(* PLC project Tc2_Utilities.GUID_TO_REGSTRING Demo, tc3-libraries-kb TwinCAT 3.1 *)
(* stored: creationDateTime 2026-05-12T10:00:00, modificationDateTime 2026-05-12T10:00:00 *)

PROGRAM P_Demo_GUID_TO_REGSTRING
  VAR
    gMachineUniqueId : GUID;  (* 从 BIOS / dongle 读到的机器唯一 ID *)
    sRegistryFormatId : STRING;  (* 写到 Windows 注册表的带花括号 GUID 串 *)
    bFormatRequest : BOOL;  (* 在线置 TRUE 触发一次格式化 *)
  END_VAR

// =============================================================================
// 场景：工业 PC 启动时把 BIOS / dongle 读到的机器唯一 ID 写到 Windows
//       注册表项 HKLM\SOFTWARE\Plant\MachineId，便于其他 Windows 服务
//       （如 OPC UA Server）通过 RegEdit 读到统一标识。
// 价值：注册表 / WMI 习惯用 '{...}' 包裹 GUID；本函数一行得到，免去
//       CONCAT('{', GUID_TO_STRING(g), '}') 三步拼接。
// 验证步骤：
//   1. 登录后 gMachineUniqueId 各字段全 0，sRegistryFormatId = ''。
//   2. 在线设置 gMachineUniqueId.Data1 := 16#12345678; .Data2 := 16#1234;
//      .Data3 := 16#5678; .Data4 := [16#9A,16#BC,16#DE,16#F0,16#12,16#34,16#56,16#78];
//   3. 写 bFormatRequest := TRUE。
//   4. 观察 sRegistryFormatId = '{12345678-1234-5678-9ABC-DEF012345678}'
//      （长度 38，含花括号，hex 大写）。
//   5. 把 gMachineUniqueId 各字段重置为 0 再触发，结果是
//      '{00000000-0000-0000-0000-000000000000}'——印证 §3 全零形态。
// =============================================================================

IF bFormatRequest THEN
    // 单次调用：永远成功，无错误码
    sRegistryFormatId := GUID_TO_REGSTRING(in := gMachineUniqueId);
    bFormatRequest := FALSE;
END_IF;
END_PROGRAM
